INTERFACE I_Robot

METHOD abort : BOOL
VAR_INPUT
END_VAR
END_METHOD

METHOD getState : eState
VAR_INPUT
END_VAR
END_METHOD

METHOD hold : BOOL
VAR_INPUT
END_VAR
END_METHOD

METHOD reset : BOOL
VAR_INPUT
END_VAR
END_METHOD

METHOD start : BOOL
VAR_INPUT
END_VAR
END_METHOD

METHOD stop : BOOL
VAR_INPUT
END_VAR
END_METHOD

END_INTERFACE

(* stored: Version 1.1.0.1, ProductVersion 3.1.4024.9
   Itf I_Robot: Id {d0cd6981-b099-45f1-a761-9ed21bd385b6}
   Method abort: Id {04b50c3f-6d7c-4d86-83c6-80516a2028e7}
   Method getState: Id {6ea73a0b-d620-4792-b9d4-dd4e241582a1}
   Method hold: Id {a93d910b-43d9-4146-8824-eb15165fbe8d}
   Method reset: Id {5148fe8d-edab-4808-801f-1de4699cedba}
   Method start: Id {1f72d0e9-602f-4e27-8f05-6ed81a0c009f}
   Method stop: Id {4c586d7f-6673-4489-8341-d5a1a853ca36} *)
